/// Implicitly generated code : DO NOT EDIT!!!
/// Checks for division by 0, if divisor is 0, replace it with 1 and report error
{attribute 'no_check' := ''}
{attribute 'check_div_real64' := ''}
FUNCTION CheckDivLReal : LREAL
VAR_INPUT
	divisor: LREAL;
END_VAR

IF divisor = 0 THEN
	// replace divisor and report error if necessary
	CheckDivLReal := 1;
	Services.fbEventHandler.Select(TC_Events.CodeEventClass.ErrorEvent)
						   .ArgSetString('div 0 LREAL')
						   .Raise();
ELSE
	CheckDivLReal:=divisor;
END_IF;

END_FUNCTION

(* stored: Version 1.1.0.1
   POU CheckDivLReal: Id {5c74c70f-78c1-464b-9a29-d100f90d2c96}, SpecialFunc None *)
